{attribute 'pack_mode' := '2'}
TYPE ST_STATION_CTRL :
STRUCT
  Cmd             : E_STATION_CTRL;
  {attribute 'displaymode':='bin'}
  nMask           : BYTE;           // nest mask for sending mover to next station
  nTargetStation  : USINT;          // where to next?
  rOffset         : REAL;           // optional offset for mover in target station when leaving sending station; 
                                    // use case: position correction of workpiece on wpc by vision
END_STRUCT
END_TYPE

(* stored: Version 1.1.0.1
   DUT ST_STATION_CTRL: Id {02617830-335f-4dc8-8bfd-38e2194b7b4d} *)
